(* IEC 61131-3 sources: eCockpitGit/test_project/src/%F%00 Library/%F%JSON, 2 files *)

(* ---- %POU%FB_JSONReader.st ---- *)
//The Initialize method must be run first
// |**Version**|**Author**| **Date** |**Changes**
// | 1         | NSN      | 04-07-20 | Creation
FUNCTION_BLOCK FB_JSONReader IMPLEMENTS ITF_StructReaderBase
VAR
//Initialize
	ready					:BOOL;				//True when the initialised method has been run
	bufferADRMax			:POINTER TO EASCII;	//The address where the file buffer ends
	bufferADROrg			:POINTER TO EASCII;	//The address where the file buffer starts
	buttomType				:EStructType;		//This saves the buttom type of the json data
	lastValueStart			:POINTER TO EASCII;
	lastValueType			:EStructType;
	lastKeyStart			:POINTER TO EASCII;
	lastKeySize				:WORD;
	treeLevel				:BYTE;				//How far down the json tree, it currently is
	treeSelectedTypes		:ARRAY[1..levelsMax] OF EStructType;
	treeSelected			:ARRAY[1..levelsMax] OF POINTER TO EASCII;
	treeSelectedArrayProg	:ARRAY[1..levelsMax] OF WORD;
END_VAR
VAR CONSTANT
	levelsMax				:BYTE:=20;
	stringMaxLen			:BYTE:=255;
END_VAR
(*%!%__DELIMITER__%!%*)

(* ---- %POU%FB_JSONWriter.st ---- *)
//This function block helps write json files, by methodising it
// |**Version**|**Author**| **Date** |**Changes**
// | 1         | NSN      | 22-06-20 | Creation
FUNCTION_BLOCK FB_JSONWriter IMPLEMENTS ITF_StructWriterBase
VAR_OUTPUT
	bufferAddress		:POINTER TO EASCII;	//The address where the file buffer starts
	bufferInvalid		:BOOL;
END_VAR
VAR
	ready				:BOOL;				//True when the initialised method has been run
	bufferPosition		:POINTER TO EASCII;	//The current address where the file is being written
	bufferMaxADR		:POINTER TO EASCII;	//The address where the file buffer ends
	treeLevel			:WORD;			//How far down the json tree, it currently is
	treeTypes			:ARRAY[1..levelsMax] OF EStructType;
	treeSingleLine		:ARRAY[1..levelsMax] OF BOOL;
	useSingleLine		:BOOL;				//Wether the JSON should be written to a single file
	bottomTypeInt		:EStructType;
	inArray				:BOOL;				//True when writing in array
	inObject			:BOOL;				//True when writing in object
	afterKey			:BOOL;				//True when just after a key
	singleVal			:BOOL;
	emptyBlock			:BOOL;
	lastComma			:POINTER TO EASCII;	//The address where the file buffer ends
END_VAR
VAR CONSTANT
	levelsMax			:BYTE:=20;
	stringMaxLen		:BYTE := 255;
END_VAR
(*%!%__DELIMITER__%!%*)
